(* IEC 61131-3 sources: park-avenue-showroom/park-avenue-showroom/000-main, 28 files *)

(* ---- 000-MAIN.ST ---- *)
VAR_GLOBAL RETAIN
  (*Light groups*)
           (*
           r1_1HallLight01                                  at %R0.0  : bool;
           r2_3LivingroomLight02_07_08                      at %R0.1  : bool; //dimm
           r3_1BalconyLight                                 at %R0.2  : bool;
           r2_2KitchenLight03                               at %R0.3  : bool;
           r2_2KitchenLight04_24                            at %R0.4  : bool;
           r2_1EatingroomLight05_06_23                      at %R0.5  : bool;
           r4_1Bedroom1Light09                              at %R0.6  : bool;
           r5_1Bedroom2Light10_22                           at %R0.7  : bool;
           r5_1Bedroom2Light11                              at %R1.0  : bool;
           r5_1Bedroom2Light12                              at %R1.1  : bool;
           r6_1WardrobeLight13_21                           at %R1.2  : bool;
           r8_1Bathroom2Light14_15_16                       at %R1.3  : bool;
           r7_1Bathroom1Light17_18_19                       at %R1.4  : bool; //dimm
           *)
           supervisorLight_01_08_23_24                      at %R0.0  : bool;
           supervisorLight_02_06_07                         at %R0.1  : bool;
           supervisorLight_balcony                          at %R0.2  : bool;
           supervisorLight_03_04                            at %R0.3  : bool;
           supervisorLight_05                               at %R0.4  : bool;
           supervisorLight_09                               at %R0.5  : bool;
           supervisorLight_10_13_22                         at %R0.6  : bool;
           supervisorLight_11_12_21                         at %R0.7  : bool;
           supervisorLight_14_16                            at %R1.0  : bool;
           supervisorLight_15                               at %R1.1  : bool;
           supervisorLight_17_19                            at %R1.2  : bool;
           supervisorLight_18                               at %R1.3  : bool;

(*Lightgroups mode switches*)
              (*
           r1_1HallLight01_auto                             at %R1.5  : bool;
           r2_3LivingroomLight02_07_08_auto                 at %R1.6  : bool; //dimm
           r2_2KitchenLight03_auto                          at %R1.7  : bool;
           r2_2KitchenLight04_24_auto                       at %R2.0  : bool;
           r2_1EatingroomLight05_06_23_auto                 at %R2.1  : bool;
           r4_1Bedroom1Light09_auto                         at %R2.2  : bool;
           r5_1Bedroom2Light10_auto                         at %R2.3  : bool;
           r5_15Bedroom2Light11_auto                        at %R2.4  : bool;
           r5_15Bedroom2Light12_auto                        at %R2.5  : bool;
           r6_1WardrobeLight13_21_auto                      at %R2.6  : bool;
           r8_1Bathroom2Light14_15_16_auto                  at %R2.7  : bool;
           r7_1Bathroom1Light17_18_19_auto                  at %R3.0  : bool; //dimm
              *)
           supervisorAuto01                                 at %R1.5  : bool; (*Hall*)
           supervisorAuto02                                 at %R1.6  : bool; (*Kitchen*)
           supervisorAuto03                                 at %R1.7  : bool; (*EatingRoom*)
           supervisorAuto04                                 at %R2.0  : bool; (*Bedroom01*)
           supervisorAuto05                                 at %R2.1  : bool; (*Livingroom*)
           supervisorAuto06                                 at %R2.2  : bool; (*Bedroom02*)
           supervisorAuto07                                 at %R2.3  : bool; (*Wardrobe*)
           supervisorAuto08                                 at %R2.4  : bool; (*Bathroom01*)
           supervisorAuto09                                 at %R2.5  : bool; (*Bathroom02*)

(*Blinds Moving Buttons*)
           r2_1EatingroomBlindsUp                           at %R3.1  : bool;
           r2_1EatingroomBlindsDown                         at %R3.2  : bool;
           r2_1EatingroomBlindsStop                         at %R3.3  : bool;
           r4_1Bedroom1BlindsUp                             at %R3.4  : bool;
           r4_1Bedroom1BlindsDown                           at %R3.5  : bool;
           r4_1Bedroom1BlindsStop                           at %R3.6  : bool;
           r5_1Bedroom2BlindsUp                             at %R3.7  : bool;
           r5_1Bedroom2BlindsDown                           at %R4.0  : bool;
           r5_1Bedroom2BlindsStop                           at %R4.1  : bool;

           generalPower                                     at %R4.2  : bool;

(*Floor Heating control*)
           floorHeatingState                                at %R4.3  : bool;

(*Water control*)
           waterState                                       at %R4.4  : bool;
           waterClose                                       at %R4.5  : bool;
           waterOpen                                        at %R4.6  : bool;
           waterAlarmReset                                  at %R4.7  : bool;
           waterAlarm                                       at %R5.0  : bool;

(*Security System*)
           security_arm                                     at %R5.1  : bool;
           security_disarm                                  at %R5.2  : bool;
           security_alarm                                   at %R5.3  : bool;
           security_alarm_reset                             at %R5.4  : bool;
           security_led                                     at %R5.5  : bool;
           security_state                                   at %R5.6  : bool;

(*TV on/off*)
             r2_3_tvOnOff                                   at %R5.7  : bool;
             r2_1_tvOnOff                                   at %R6.0  : bool;

(*Update*)
             updateIridiumProjectFlag                       at %R6.1  : bool;

(*Dimmed groups brightness level*)
           r2_3LivingroomLight02_07_08_level                at %R105  : real;
           r7_1Bathroom1Light17_18_19_level                 at %R109  : real;

(*Blinds position control*)
           r2_1EatingroomBlindsPosition                     at %R113   : real;
           r4_1Bedroom1BlindsPosition                       at %R117   : real;
           r5_1Bedroom2BlindsPosition                       at %R121   : real;

(*Floor Heating control*)
           floorHeatingLevel                                at %R125   : real;

(*AC set temperature*)
           r2_3_GuestRoomACSetTemperature                   at %R129   : real;
           r5_Bedroom2ACSetTemperature                      at %R133   : real;
           r4_Bedroom1ACSetTemperature                      at %R140   : real;
(*AC mode*)
           r2_3_GuestRoomACMode                             at %R137   : usint;
           r5_Bedroom2ACMode                                at %R138   : usint;
           r4_Bedroom1ACMode                                at %R139   : usint;

END_VAR

VAR_GLOBAL CONSTANT
  new : BOOL := false;
  AUTO_MODE_DEFAULT_STATE   : bool := true;
  AUTO_MODE_DEFAULT_TIME    : time := t#150s;
END_VAR

(* ---- fbBlindController.ST ---- *)
FUNCTION_BLOCK fbBlindController
  VAR_INPUT
    timeTo_up_down : time;
    open           : bool r_edge;
    close          : bool r_edge;
    stop           : bool r_edge;
    setPosition    : real;
  END_VAR
  VAR_OUTPUT
    up             : bool;
    down           : bool;
    currentPosition: real:=100;
  END_VAR
  VAR_IN_OUT

  END_VAR
  VAR
    t1             : time;
    timer          : fbTimer;
    direction      : bool;    (*True - UP, False - DOWN*)
    position       : real:=100;
    stopTtigg      : r_trig;
    openTrigg      : r_trig;
    closeTrigg     : r_trig;
  END_VAR
  VAR_TEMP

  END_VAR

  timer();
  if timer.isRun then
    if direction then
      position := position + ((time_to_real(timer.currentTime - t1)/10.)/
                              (time_to_real(timeTo_up_down)/1000.));
    else
      position := position - ((time_to_real(timer.currentTime - t1)/10.)/
                              (time_to_real(timeTo_up_down)/1000.));
    end_if;
    t1 := timer.currentTime;
  else
    t1 := t#0ms;
  end_if;

  currentPosition := position;

  if setPosition>0. then
     if setPosition>currentPosition then
        open:=true;
     end_if;
     if setPosition<currentPosition then
        close:=true;
     end_if;
  end_if;

  if currentPosition <= 0. or currentPosition >= 100. then
     stop:= true;
  end_if;

  if abs(setPosition - currentPosition) <= 0.05 then
     setPosition:=0.;
     stop:= true;
  end_if;

  openTrigg(CLK := open);
  if openTrigg.Q then
    timer(start := true, timeToCount := timeTo_up_down + t#20ms);
    t1 := t#0ms;
    up := true;
    down := false;
    direction := true;
  end_if;

  closeTrigg(CLK := close);
  if closeTrigg.Q then
    timer(start := true, timeToCount := timeTo_up_down + t#20ms);
    t1 := t#0ms;
    up := false;
    down := true;
    direction := false;
  end_if;

  stopTtigg(CLK := stop);
  if stopTtigg.Q then
     up:=false;
     down:=false;
     timer(reset:=true);
     setPosition:=0.;
  end_if;

  timer();
  if timer.isDone then
    timer(reset := true);
    up := false;
    down := false;
  end_if;
END_FUNCTION_BLOCK

(* ---- fbBoolObserver.ST ---- *)
FUNCTION_BLOCK fbBoolObserver
  VAR_INPUT
	  state        : bool;
  END_VAR
  VAR
      prevState : bool;
  END_VAR
  VAR_OUTPUT
      stateChanged : bool;
      rising       : bool;
      falling      : bool;
  END_VAR
  VAR_IN_OUT

  END_VAR
  VAR_TEMP

  END_VAR
      stateChanged := false;
      rising       := false;
      falling      := false;
      if state <> prevState then
         stateChanged := true;
         if state then
            rising := true;
         else
            falling := true;
         end_if;
         prevState := state;
      end_if;
END_FUNCTION_BLOCK

(* ---- fbDataKeeper.st ---- *)
VAR_GLOBAL
    //reader : ReadFromFile; {hidden}
    //writer : WriteToFile;  {hidden}
END_VAR

FUNCTION_BLOCK fbSaveData  {hidden}
  VAR_INPUT
      save     : bool r_edge;
  END_VAR
  VAR_OUTPUT
      idle        : bool := true;
      done        : bool ;
      currentFile : string[20];
  END_VAR
  VAR_IN_OUT
      fullPath    : string[20];
      dataSize    : udint;
      data        : udint;
  END_VAR
  VAR
      lastError: string;
      writer   : WriteToFile;  {hidden}
  END_VAR
  VAR_TEMP
  END_VAR

  done    := false;

  if save then
     idle := false;
     save := false;
  end_if;

  writer( fileName := fullPath,
          srcVar   := data,
          exec     := not idle,
          seek     := 0,
          size     := dataSize);

  if writer.done then
     idle := true;
     done := true;
  end_if;

  if GetLastErr() <> 0 then
     GetLastErrTxt(errCode := GetLastErr(), errMessage := lastError);
  end_if;

  currentFile := fullPath;

END_FUNCTION_BLOCK

FUNCTION_BLOCK fbLoadData  {hidden}
  VAR_INPUT
      load     : bool r_edge;
  END_VAR
  VAR_OUTPUT
      idle        : bool := true;
      done        : bool;
      currentFile : string[20];
  END_VAR
  VAR_IN_OUT
      fullPath    : string[20];
      dataSize : udint;
      data     : udint;
  END_VAR
  VAR
      lastError: string;
      reader   : ReadFromFile; {hidden}
  END_VAR
  VAR_TEMP
  END_VAR

  done    := false;

  if load then
     idle := false;
     load := false;
  end_if;

  reader( fileName := fullPath,
          dstVar   := data,
          exec     := not idle,
          seek     := 0,
          size     := dataSize);

  if reader.done then
     idle := true;
     done := true;
  end_if;

  if GetLastErr() <> 0 then
     GetLastErrTxt(errCode := GetLastErr(), errMessage := lastError);
  end_if;

  currentFile := fullPath;

END_FUNCTION_BLOCK

VAR_GLOBAL RETAIN
    dataSaver  :fbSaveData;    {hidden}
    dataLoader :fbLoadData;    {hidden}
END_VAR

FUNCTION_BLOCK fbDataKeeper
  VAR_INPUT
      path     : string[10];
      fileName : string[10];
      dataSize : udint;
  END_VAR
  VAR_OUTPUT
      load     : bool;
  END_VAR
  VAR_IN_OUT
      data       : udint;
  END_VAR
  VAR
      save     : bool;
      fullPath : string[20];
      init     : bool;
  END_VAR
  VAR_EXTERNAL
      at %s20.3 : bool;
  END_VAR

      fullPath := '/'+ path + '/' +fileName;

      if not init then
         if not FileExists(fileName := fullPath) then
            if not FileExists(fileName := path) then
               DirCreate(dirName := path);
            end_if;
            load := true;
         end_if;
         init := true;
      end_if;

      if not load  then
         if dataLoader.idle then
            dataLoader( load     := true,
                        fullPath := fullPath,
                        dataSize := dataSize,
                        data     := data);
         end_if;
         if dataLoader.done and dataLoader.currentFile = fullPath then
            load := true;
         end_if;
      end_if;

      if %S20.3 and init and load then
         save := true;
      end_if;

      if dataSaver.idle and save  then
         dataSaver( save      := true,
                    fullPath  := fullPath,
                    dataSize  := dataSize,
                    data      := data);
      end_if;
      if dataSaver.done and dataSaver.currentFile = fullPath then
         save     := false;
      end_if;

      dataSaver (data:=data, fullPath := fullPath, dataSize := dataSize);
      dataLoader(data:=data, fullPath := fullPath, dataSize := dataSize);

END_FUNCTION_BLOCK

(* ---- fbFloorHeatingSimple.ST ---- *)
FUNCTION_BLOCK fbFloorHeatingSimple
  VAR_INPUT
       period : time := t#30m;
  END_VAR
  VAR_OUTPUT
      out : bool;
  END_VAR
  VAR_IN_OUT
       state : bool;
       power : real;
  END_VAR
  VAR
       pwmGenerator : PWM;
  END_VAR
  VAR_TEMP
  END_VAR

       pwmGenerator(Enb := true, Per := period, Pls := power, Out =>  out);

       if state then
          out := pwmGenerator.Out;
       else
          out := false;
       end_if;

END_FUNCTION_BLOCK

(* ---- fbGlobalCacheSender.ST ---- *)
TYPE
  irCodesString   :  array[100..150] of string[255];
END_TYPE

FUNCTION_BLOCK fbGlobalCacheSender
  VAR_INPUT
      sendCode : uint;
      channel  : uint;
  END_VAR
  VAR_IN_OUT
      codes   : irCodesString;
  END_VAR
  VAR
      tcpSender : fbSendTo;
      code      : string[255];
      send      : bool;
  END_VAR
      if sendCode <> 0 and (not send) then
         code := codes[sendCode];
         code := code + '$R';
         send           := true;
         sendCode := 0;
      end_if;

      if send then

          tcpSender( chanCode := channel,
                     rq       := not tcpSender.mesSent,
                     lenTx    := len(code),
                     data     := void(code));

          if tcpSender.mesSent then
             send         := false;
          end_if;
      end_if;
END_FUNCTION_BLOCK

(* ---- fbPanel.ST ---- *)
FUNCTION_BLOCK fbPanel
  VAR_INPUT
      button : array[1..6] of fbButtonProcessor;
  END_VAR
  VAR_OUTPUT
      led : array[1..6] of bool;
  END_VAR
  VAR_IN_OUT
  END_VAR
  VAR
  END_VAR
  VAR_TEMP
  END_VAR

    button[1]();
    button[2]();
    button[3]();
    button[4]();
    button[5]();
    button[6]();

END_FUNCTION_BLOCK

(* ---- fbRealObserver.ST ---- *)
FUNCTION_BLOCK fbRealObserver
  VAR_INPUT
	  value        : real;
  END_VAR
  VAR
      prevValue : real;
  END_VAR
  VAR_OUTPUT
      valueChanged : bool;
      rising       : bool;
      falling      : bool;
  END_VAR
      valueChanged := false;
      rising       := false;
      falling      := false;

      if value <> prevValue then
         valueChanged := true;
         if value > prevValue then
            rising := true;
         else
            falling := true;
         end_if;
         prevValue := value;
      end_if;
END_FUNCTION_BLOCK

(* ---- fbSecuritySystem.ST ---- *)
Type
    SecuritySystemState : (init, disarmed, arming, armed, alarming);
    SecurityZoneMode    : (NO,NC);
    SecurityConfig      :
        struct
               exitTime        :time := t#15s;
               enterenceTime   :time := t#15s;
               Z1Mode          :SecurityZoneMode := NC;
               Z2Mode          :SecurityZoneMode := NC;
               Z3Mode          :SecurityZoneMode := NC;
               Z4Mode          :SecurityZoneMode := NC;
               Z5Mode          :SecurityZoneMode := NC;
               KeyBoardEnable  :bool := false;
               KeyBImpulseTime :time := t#1s;
        end_struct;
end_type

FUNCTION_BLOCK fbSecuritySystem
(*
Error codes description:
1 - Can't Armed system because Sabotage alarm is on.
2 - Can't Armed system because one or more zone is broken.
3 - Keypad error.
*)
  VAR_INPUT
    config      :SecurityConfig;
    Z1          :bool; (*Enter/Exit Door.*)
    Z2          :bool; (*Enter/Exit Zone.*)
    Z3          :bool; (*Doors, windows and PIR sensors.*)
    Z4          :bool; (*Other sensors.*)
    Z5          :bool; (*Tamper zone.*)
    keyBoard    :bool; (*relay keypad contact.*)
    arm         :bool r_edge;  (*Security On flag.*)
    disarm      :bool r_edge;  (*Security Off flag.*)
    alarmReset  :bool r_edge;  (*Alarm reset flag.*)
    sabotageReset:bool r_edge; (*Reset sabotege alarm.*)
  END_VAR
  VAR_OUTPUT
    securityState :bool;      (*TRUE when systen armed.*)
    alarm         :bool;      (*Alarm flag.*)
    siren         :bool;      (**)
    ledIndicator  :bool;      (**)
    sabotage      :bool;      (*TRUE when tamper zone was broken until reset by sabotageReset variable.*)
    error         :bool;      (*TRUE when error until next cycle.*)
    errorCode     :usint;     (*Error descrintion code.*)
  END_VAR
  VAR
    state               :SecuritySystemState;
    keyBoardImpulse     :TP;
    keyBoardEvent       :f_trig;
    keyBoardImpulseEnd  :f_trig;
    exitTimer           :ton;
    entranceTimer       :ton;
    ledPulse            :PWM;
    userEnterPassword   :bool;
    armWithoutDelay     :bool;
  END_VAR

//--Zone inverting accordin to their mode (FALSE - normal state)--//
  if config.Z1Mode = NC then
     Z1 := not Z1;
  end_if;

  if config.Z2Mode = NC then
     Z2 := not Z2;
  end_if;

  if config.z3Mode = NC then
     z3 := not z3;
  end_if;

  if config.z4Mode = NC then
     z4 := not z4;
  end_if;

  if config.z5Mode = NC then
     z5 := not z5;
  end_if;

//--General process-//
  if state <> init then
      error := false;

      if config.KeyBoardEnable then
          keyBoardImpulse(IN := not keyBoard, PT := config.KeyBImpulseTime + t#1s);
          keyBoardEvent(CLK := not keyBoard);
          keyBoardImpulseEnd(CLK := keyBoardImpulse.Q);

          userEnterPassword := false;
          userEnterPassword := keyBoardEvent.Q and keyBoardImpulse.Q;

          if keyBoardImpulseEnd.Q and (not keyBoard) then
             error     := true;
             errorCode := 3;
          end_if;
      end_if;

      if Z5 then
         sabotage := true;
      else
         if sabotageReset then
            sabotage := false;
         end_if;
      end_if;
  end_if;

  case state of
    init:
        state := disarmed;

    disarmed:
        if userEnterPassword or arm then
           if (not Z3) and (not Z4) and  (not Z5) and (not sabotage) then
              state := arming;
              if arm then
                 armWithoutDelay := true;
              else
                 armWithoutDelay := false;
              end_if;
           else
              error     := true;
              if sabotage then
                 errorCode := 1;
              else
                 errorCode := 2;
              end_if;
           end_if;
        end_if;
        ledIndicator := false;
        siren        := false;

    arming:
        exitTimer(IN := true, PT := config.exitTime);

        if Z3 or Z4 or Z5 then
           exitTimer(IN := false);
           error     := true;
           if sabotage then
              errorCode := 1;
           else
              errorCode := 2;
           end_if;
           state     := disarmed;
        end_if;

        if exitTimer.Q or armWithoutDelay then
           exitTimer(IN := false);
           if (not Z1) and (not Z2) then
              state := armed;
           else
              error     := true;
              errorCode := 2;
              state     := disarmed;
           end_if;
        end_if;

        ledPulse(Enb := true, Per := t#1s, Pls := 50.0, Out => ledIndicator);

    armed:
        if Z1 then
           entranceTimer.IN := true;
        end_if;

        if (Z2 and not entranceTimer.IN) or Z3 or Z4 or Z5 then
           state := alarming;
        end_if;

        //if (userEnterPassword and entranceTimer.IN) or disarm then
        if userEnterPassword or disarm then
           state := disarmed;
           entranceTimer(IN := false);
        end_if;

        entranceTimer(PT := config.enterenceTime);
        if entranceTimer.Q then
           entranceTimer(IN := false);
           state := alarming;
        end_if;

        if entranceTimer.IN then
           ledPulse(Enb := true, Per := t#1s, Pls := 50.0, Out => ledIndicator);
        else
           ledIndicator := true;
        end_if;
        siren := false;

    alarming:
        siren := true;
        ledPulse(Enb := true, Per := t#2s, Pls := 75.0, Out => ledIndicator);
        if alarmReset then
           state := armed;
        end_if;

        if userEnterPassword or disarm then
           state := disarmed;
           entranceTimer(IN := false);
        end_if;

  end_case;

  if state <> init then
       if state = alarming then
         alarm := true;
      else
         alarm := false;
      end_if;

      if state = armed then
         securityState := true;
      end_if;

      if state = disarmed then
         securityState := false;
      end_if;
  end_if;

END_FUNCTION_BLOCK

(* ---- fbTimer.ST ---- *)
FUNCTION_BLOCK fbTimer
  VAR_INPUT
      start      : bool r_edge;
      reset      : bool r_edge;
      timeToCount: time;
  END_VAR
  VAR_OUTPUT
      isRun : bool;
      isDone: bool;
      currentTime : time;
  END_VAR
  VAR_IN_OUT
  END_VAR
  VAR
      timer: TON;
  END_VAR
  VAR_TEMP
  END_VAR

         if start and not isRun then
            timer.IN := true;
            start    := false;
            isRun    := true;
            isDone   := false;
            timer.PT := timeToCount;
         end_if;

         if start and isRun then
            timer(IN :=false);
            timer(IN :=true);
         end_if;

         if isRun then
            timer();
            if timer.ET>=timer.PT then
               isDone:=true;
               isRun :=false;
               timer.IN:=false;
               timer();
            end_if;
         end_if;

         if reset then
            timer.IN:=false;
            isDone:=false;
            isRun:=false;
            timer();
         end_if;

         timer();
         currentTime:=timer.ET;
END_FUNCTION_BLOCK

(* ---- prgNotifications.ST ---- *)
FUNCTION_BLOCK fbBoolObserver
  VAR_INPUT
      in : bool;
  END_VAR
  VAR
      prevState : bool;
  END_VAR
  VAR_OUTPUT
      stateChanged : bool;
      state        : bool;
      rising       : bool;
      falling      : bool;
  END_VAR
      stateChanged := false;
      rising       := false;
      falling      := false;
      state        := in;
      if state <> prevState then
         stateChanged := true;
         if state then
            rising := true;
         else
            falling := true;
         end_if;
         prevState := state;
      end_if;
END_FUNCTION_BLOCK

FUNCTION_BLOCK fbRealObserver
  VAR_INPUT
      in : ptr_to real;
  END_VAR
  VAR
      prevValue : real;
  END_VAR
  VAR_OUTPUT
      valueChanged : bool;
      value        : real;
      rising       : bool;
      falling      : bool;
  END_VAR
      valueChanged := false;
      rising       := false;
      falling      := false;
      value        := in^;

      if value <> prevValue then
         valueChanged := true;
         if value > prevValue then
            rising := true;
         else
            falling := true;
         end_if;
         prevValue := value;
      end_if;
END_FUNCTION_BLOCK

(* ---- RalayAndDimmer.ST ---- *)
type
    motionSensorMode: (null, NO, NC);
    doorSensorMode:   (null, NO, NC);
    motionSensor:
        struct
            state:bool;
            mode :motionSensorMode;
        end_struct;
    doorSensor:
        struct
            state:bool;
            mode :doorSensorMode;
        end_struct;
end_type

FUNCTION_BLOCK fbAutoRelay
  VAR_IN_OUT
           //trigButton      : bool ;                  (**)
           //autoMode        : bool :=true;
  END_VAR
  VAR_INPUT
           Sensor_Door      : doorSensor;   (**)
           Sensor_Motion    : motionSensor; (**)

           autoMode      : bool ;                    (**)
           nightMode     : bool ;                    (**)

           forgetMode    : bool :=false;             (**)

           anyLightOn             : bool ;           (**)
           anyLightChanged        : bool ;           (**)

           timeAfterDoorOpenClose : time :=t#1m;     (**)
           timeAfterMotionDetect  : time :=t#10m;     (**)
           timeAfterLastAction    : time :=t#1m;     (**)
           setState               : bool ;           (**)
  END_VAR
  VAR_OUTPUT
           personLeft   : bool ;                     (**)
           forget       : bool ;                     (**)
           stateChanged : bool ;                     (**)
           state        : bool ;                     (**)
  END_VAR
  VAR
           timerAfterDoorOpened     : fbTimer;
           timerAfterDoorClosed     : fbTimer;
           timerAfterMotionDetected : fbTimer;
           timerAfterLastAction     : fbTimer;

           doorSensRise        : r_trig;
           doorSensFall        : f_trig;
           doorClosed          : bool;
           doorOpened          : bool;
           motionSensRise      : r_trig;
           motionSensFall      : f_trig;
           motionDetected      : bool;
           motionEnd           : bool;
           nightModeOff        : f_trig;
  END_VAR

        (*Refresh outputs.*)
        stateChanged:=false;
        personLeft  :=false;
        forget      :=false;

        nightModeOff(CLK := nightMode);
        if nightModeOff.Q then
           timerAfterDoorOpened    (reset := true);
           timerAfterDoorClosed    (reset := true);
           timerAfterMotionDetected(reset := true);
           if autoMode then
              setState:=false; end_if;
        end_if;

        (*Auto*)
        if autoMode and nightMode then
           (*Process move sensor.*)
           motionSensRise(CLK := Sensor_Motion.state);
           motionSensFall(CLK := Sensor_Motion.state);
           case Sensor_Motion.mode of
                NO:
                   motionDetected := motionSensRise.Q;
                   motionEnd      := motionSensFall.Q;
                NC:
                   motionDetected := motionSensFall.Q;
                   motionEnd      := motionSensRise.Q;
           end_case;
           (*Process door sensor.*)
           case Sensor_Door.mode of
                NO:
                   doorSensRise(CLK := Sensor_Door.state, Q => doorOpened);
                   doorSensFall(CLK := Sensor_Door.state, Q => doorClosed);
                NC:
                   doorSensRise(CLK := Sensor_Door.state, Q => doorClosed);
                   doorSensFall(CLK := Sensor_Door.state, Q => doorOpened);
           end_case;
           (*Timers process.*)
           timerAfterDoorOpened     (timeToCount :=timeAfterDoorOpenClose);
           timerAfterDoorClosed     (timeToCount :=timeAfterDoorOpenClose);
           timerAfterMotionDetected (timeToCount :=timeAfterMotionDetect);
           (*Door opened/closed logic.*)
           (*Door opened.*)
           if doorOpened and not anyLightOn then
              setState:=true;
              timerAfterDoorOpened( start := true);
           end_if;
           timerAfterDoorOpened();
           if timerAfterDoorOpened.isDone then
              setState :=false;
              timerAfterDoorOpened(reset := true);
           end_if;
           (*Door closed.*)
           if doorClosed then
              timerAfterDoorClosed( start := true);
           end_if;
           if timerAfterDoorClosed.isDone then
              setState  :=false;
              personLeft:=true;
              timerAfterDoorClosed(reset := true);
           end_if;
           (*Motion detecion logic.*)
           (*Motion detected.*)
           if motionDetected then
              if not anyLightOn then
                 setState := true;
//                 timerAfterMotionDetected(start := true);
              end_if;
              timerAfterDoorOpened    (reset := true);
              timerAfterDoorClosed    (reset := true);
           end_if;
           (*Motion end.*)
           if motionEnd then
              timerAfterMotionDetected(start := true);
           end_if;
           if timerAfterMotionDetected.isDone then
              setState:=false;
              timerAfterMotionDetected(reset := true);
           end_if;
        end_if;

        (*Forget mode.*)
        if forgetMode then
           timerAfterLastAction(timeToCount := timeAfterLastAction);
           if motionDetected then
              timerAfterLastAction(start := true);
           end_if;
           if timerAfterLastAction.isDone then
              timerAfterLastAction(reset:=true);
              forget:=true;
           end_if;
           if anyLightChanged then
              timerAfterLastAction(reset:=true);
              timerAfterLastAction(start:=true);
           end_if;;
        end_if;

        (*Set state.*)
        if setState<>state then
           stateChanged:= true;
           state       := setState;
        end_if;
END_FUNCTION_BLOCK

FUNCTION_BLOCK fbManualRelay
  VAR_IN_OUT
           trigButton          : bool ; (*Button for trigger control.*)
  END_VAR
  VAR_INPUT
           setState            : bool ; (*Turn on/off channel.*)
  END_VAR
  VAR
           trigButtonOff   : f_trig;
           trigButtonOn    : r_trig;
  END_VAR
  VAR_OUTPUT
           stateChanged : bool  ;           (*State changed flag.    *)
           state        : bool ;            (*Current state of relay.*)
  END_VAR
        (*Refresh outputs.*)
        stateChanged:=false;

        trigButtonOn (CLK := trigButton);
        trigButtonOff(CLK := trigButton);

        if trigButtonOn.Q  then
           setState:=true;
        end_if;

        if trigButtonOff.Q then
           setState:=false;
        end_if;

        if setState<>state then
           stateChanged := true;
           state        := setState;
           trigButton   := state;
        end_if;

END_FUNCTION_BLOCK

function_block fbButtonProcessor
    var_input
        btn          :  bool; (*Pointer to Button*)
        longPressTime: time := t#1000ms;       (*Long press time detect.*)
    end_var
    var_in_out
    end_var
    var_output
        longPress  :bool;                     (*Long press flag.*)
        shortPress :bool;                     (*Short press flag.*)
        btnPressed :bool;                     (*Event flag on button pressed.*)
        btnReleased:bool;                     (*Event flag on button released.*)
        btnState   :bool;                     (*Button state.*)
        longPressAndHold:bool;                (*Long press and hold flag.*)
    end_var
    var
        btnPrevState  :bool;
        timer         :fbTimer;
    end_var
    var
    end_var
        (*Refresh outputs.*)
        longPress  :=false;
        shortPress :=false;
        btnPressed :=false;
        btnReleased:=false;
        btnState   :=btn;
        (*Button event detection.*)
        timer(timeToCount := longPressTime);
        if btn <> btnPrevState then
           (*Button status changed.*)
           btnPrevState := btn;
           if btn then
              (*Button pressed.*)
              btnPressed:=true;
              if not timer.isRun then
                 timer.start:=true;
                 timer();
              end_if;
           else
              (*Button Released.*)
              btnReleased:=true;
              if timer.isRun then
                 timer.reset := true;
                 timer();
                 shortPress:=true;
              end_if;
           end_if;
        end_if;
        if timer.isDone then
           (*Time out.*)
           timer.reset := true;
           timer();
           longPress:=true;
        end_if;

        if longPress then
           longPressAndHold:=true;
        end_if;

        if btnReleased then
           longPressAndHold := false;
        end_if;

end_function_block

function_block fbManualDimm
    var_input
        btn      : bool;                       (*Pointer to button processor.*)
        minValue : real:=20.0;                 (*Minimum value of channel.*)
        maxValue : real:=100.0;                (*Maximum value of channel.*)
        dimmSpeed: real:=25.0;                 (*Up/Down dimming speed, %/sec.*)
        setValue : real;                       (**)
        setState : bool;                       (*Turn on/off channel like relay. Set to levels like short press.*)
    end_var
    var_in_out
        slider    :real;                       (*Slider in % in range from minValue to maxValue.*)
        trigButton:bool;                       (*Button for trigger contol.*)
    end_var
    var_output                                 (*Current value of channel.*)
        value       :real;
        valueChanged:bool;
        state       :bool;
        stateChanged:bool;
    end_var
    var
        direction :real:=1.0;
        userValue :real;
        dimming   :bool;
        timer     :TON;
        cycleTime :time;
        prevTime  :time;
        step      :real;
        init      :bool;
        prevValue :real;
        prevSetValue:real;
        prevSlider:real;
        buttonProcessor : fbButtonProcessor;
    end_var
    var_temp

    end_var
        (*Init block.*)
        if not init then
           init:=true;
           userValue:=maxValue;
        end_if;

        buttonProcessor(btn := btn);

        (*Calc 1% in current range.*)
        if minValue<20. then
           minValue:=20.; end_if;
        step:=((maxValue-minValue)/100.);

        (*Reset outputs.*)
        valueChanged:=false;
        stateChanged:=false;

        (*Set value by setValue variable.*)
        if setValue<>prevSetValue then
           if setValue=0.0 then
              value:=0.0;
           elsif setValue=1.0 then
              value := minValue;
           else
              value := minValue + (step*setValue);
           end_if;
        end_if;

        (*Set value by slider.*)
        if slider<>prevSlider then
           if slider=0.0 then
              value:=0.0;
           elsif slider=1.0 then
              value := minValue;
           else
              value := minValue + (step*slider);
           end_if;
        end_if;

        (*On/Off channel.*)
        (*On/Off by impulse button.*)
        if buttonProcessor.shortPress then
           if value >= minValue then
              userValue := value;
              value  := 0.0;
           else
              value := userValue;
           end_if;
        end_if;
        (*On/Off by setState variable.*)
        if setState<>state then
           if setState then
              value:=userValue;
           else
              value:=0.0;
           end_if;
        end_if;
        (*On/Off by triggButton variable.*)
        if trigButton <> state then
           if trigButton then
              value:=userValue;
           else
               value:=0.0;
           end_if;
        end_if;

        (*Dimming.*)
        timer(IN := buttonProcessor.longPressAndHold , PT := t#100s);
        cycleTime:=SUB_TIME(IN1 := timer.ET, IN2 := prevTime);
        prevTime:=timer.ET;

        if buttonProcessor.longPressAndHold then
           dimming:=true;
           value:=value + (direction * (step * dimmSpeed * (TIME_TO_REAL(cycleTime)/1000.)));
           if value > maxValue then
              value := maxValue; end_if;
           if value < minValue then
              value := minValue; end_if;
        end_if;

        (*End_dimming.*)
        if dimming and buttonProcessor.btnReleased then
           dimming   := false;
           direction := direction*(-1.0);
           userValue := value;
        end_if;

         (*Update slider and local variables.*)
         if value=0.0 then
            slider:=0.0;
         elsif value=minValue then
            slider:=1.0;
         else
            slider:=((value-minValue)/step);
            if slider>100. then
               slider:=100.; end_if;
         end_if;
         prevSlider  :=slider;
         setValue    :=slider;
         prevSetValue:=slider;
         trigButton  := REAL_TO_BOOL(value);
         setState    := trigButton;

         (*Update outputs.*)
         if state <> REAL_TO_BOOL(value) then
            stateChanged:=true;
            state := REAL_TO_BOOL(value);
         end_if;
         if value <> prevValue then
            prevValue    :=value;
            valueChanged :=true;
         end_if;
end_function_block

(* ---- WaterLeakegeControl.ST ---- *)
TYPE
  WaterSensorModeType : (NO, NC); (*NO: Alarm when input is TRUE. NC: alarm when input is FALSE.*)
  WaterValveModeType  : (NO, NC); (*NO: Valve is open when output = FALSE; NC: Valve is open when output = TRUE *)
  WaterLeakegeControlConfig:
    STRUCT
      sensorMode                : WaterSensorModeType := NO;
      valveMode                 : WaterValveModeType  := NO;
      timeTreshold              : time           := t#5s;
      waterOnSendorsTimeoutTime : time           := t#10m;
    END_STRUCT;
END_TYPE

FUNCTION_BLOCK fbWaterLeakegeControl
  VAR_INPUT
  //--Inputs--//
      sensor     : bool ;                     (*Water Leakege Sensor.*)
  //--Commands--//
      openWater  : bool r_edge;               (*Flag to open water if it possible.*)
      closeWater : bool r_edge;               (*Flag to close water.*)
      alarmReset : bool r_edge;               (*Flag to reset alarm.*)
  //--Configuration variables--//
      config     : WaterLeakegeControlConfig; (*Zone configuration.*)
      autoControl: bool := true;
  END_VAR
  VAR_OUTPUT
      valve      : bool;                      (*Valve.*)
      alarm      : bool;                      (*True when water was closed by sensor until not reset.*)
  END_VAR
  VAR_IN_OUT
      waterState : bool                       (*TRUE = Water is open.*);
  END_VAR
  VAR
      waterOnSensor         : bool;
      timeTreshold          : ton;
      waterOnSendorsTimeout : tp;
      timeOut               : f_trig;
  END_VAR

  case config.sensorMode of
       NO: waterOnSensor := sensor;
       NC: waterOnSensor := not sensor;
  end_case;

  if openWater then
     waterState := true;
  end_if;

  if closeWater then
     waterState := false;
  end_if;

  if alarmReset then
     alarm := false;
     waterOnSendorsTimeout(IN := false); // timer call to reset
     waterOnSendorsTimeout.IN := true;
  end_if;

  timeTreshold(IN := waterOnSensor, PT := config.timeTreshold);
  waterOnSendorsTimeout(PT := config.waterOnSendorsTimeoutTime);
  timeOut(CLK := waterOnSendorsTimeout.Q);

  if timeTreshold.Q or (timeOut.Q and waterOnSensor) then
     alarm := true;
  end_if;

  if alarm and autoControl then
     waterState := false;
  end_if;

  if waterState and alarm then
     waterState := false;
  end_if;

  case config.valveMode of
       NO: valve := not waterState;
       NC: valve := waterState;
  end_case;

END_FUNCTION_BLOCK

(* ---- prgBalconyLight.ST ---- *)
PROGRAM prgBalconyLight
  VAR_INPUT
  END_VAR
  VAR_OUTPUT
  END_VAR
  VAR
      Lamp1     : fbManualRelay;

      button    : fbButtonProcessor;

      init      : bool;
  END_VAR
  VAR_TEMP
  END_VAR

  if not init then
     init := true;
  end_if;

  button(btn :=button_04_1);

  if button.shortPress then
     Lamp1.setState:= not Lamp1.state;
  end_if;

  lamp1(
        trigButton := supervisorLight_balcony,
        state      => light_balcony
        );

  if generalPowerObserver.falling then
     Lamp1.setState := false;
  end_if;

END_PROGRAM

(* ---- prgBathroom1Light.ST ---- *)
PROGRAM prgBathroom1Light
  VAR_INPUT
  END_VAR
  VAR_OUTPUT
  END_VAR
  VAR

      Lamp1,
      Lamp2     : fbManualRelay;

      Auto8      : fbAutoRelay;

      button1,
      button2   : fbButtonProcessor;

      init      : bool;

  END_VAR
  VAR_TEMP
  END_VAR

  if not init then
     supervisorAuto08                 := AUTO_MODE_DEFAULT_STATE;
     Auto8.timeAfterMotionDetect       := AUTO_MODE_DEFAULT_TIME;
     Auto8.Sensor_Motion.mode          := NC;
     Auto8.nightMode                   := true;

     init := true;
 end_if;

 (*Lamp1*)
  button1(btn := button_15_1_16_1);

  if button1.shortPress then
     Lamp1.setState := not Lamp1.state;
  end_if;

  Lamp1(trigButton := supervisorLight_17_19);

  light_17_19_level := BOOL_TO_REAL(Lamp1.state) * 100.;

  Auto8(Sensor_Motion.state   := msensor08,
        autoMode              := supervisorAuto08);

  if Auto8.stateChanged then
     Lamp1.setState := Auto8.state;
  end_if;

  (*Lamp2*)
  button2(btn := button_15_2_16_2);

  if button2.shortPress then
     Lamp2.setState := not Lamp2.state;
  end_if;

  Lamp2(trigButton := supervisorLight_18);

  light_18_mirror := Lamp2.state;

  if generalPowerObserver.falling then
     Lamp1.setState := false;
     Lamp2.setState := false;
  end_if;

END_PROGRAM

(* ---- prgBathroom2Light.ST ---- *)
PROGRAM prgBathroom2Light
 VAR_INPUT
  END_VAR
  VAR_OUTPUT
  END_VAR
  VAR
      Lamp1,
      Lamp2     : fbManualRelay;

      Auto9     : fbAutoRelay;

      button1,
      button2   : fbButtonProcessor;

      init      : bool;

      //kostyl    :R_TRIG;

  END_VAR
  VAR_TEMP
  END_VAR

  if not init then
     supervisorAuto09                  := AUTO_MODE_DEFAULT_STATE;
     Auto9.timeAfterMotionDetect       := AUTO_MODE_DEFAULT_TIME;
     Auto9.Sensor_Motion.mode          := NC;
     Auto9.nightMode                   := true;

     init := true;
 end_if;

 (*Lamp1*)
  button1(btn := button_20_1_21_1);

  if button1.shortPress then
     Lamp1.setState := not Lamp1.state;
  end_if;

  //эта штука появилась тут из-за того, что нужно было
  //добавить в сценарий "пришел домой" включение света в СУ2
  //а Юрко не нашел кода, который этот сценарий реализует
  //kostyl(CLK := generalPower);
  if generalPowerObserver.rising Then
     supervisorLight_14_16 := true;
  End_if;

  Lamp1(trigButton := supervisorLight_14_16);

  light_14_16 := Lamp1.state;

  Auto9(Sensor_Motion.state   := msensor09,
        autoMode              := supervisorAuto09);

  if Auto9.stateChanged then
     Lamp1.setState := Auto9.state;
  end_if;

  (*Lamp2*)
  button2(btn := button_20_2_22_1);

  if button2.shortPress then
     Lamp2.setState := not Lamp2.state;
  end_if;

  Lamp2(trigButton := supervisorLight_15);

  light_15 := Lamp2.state;

  if generalPowerObserver.falling then
     Lamp1.setState := false;
     Lamp2.setState := false;
  end_if;

END_PROGRAM

(* ---- prgBedroom1Light.ST ---- *)
PROGRAM prgBedroom1Light
  VAR_INPUT
  END_VAR
  VAR_OUTPUT
  END_VAR
  VAR
      Lamp1     : fbManualRelay;

      Auto4      : fbAutoRelay;

      button    : fbButtonProcessor;

      init      : bool;
  END_VAR
  VAR_TEMP
  END_VAR

  if not init then

     supervisorAuto04                := AUTO_MODE_DEFAULT_STATE;
     Auto4.timeAfterMotionDetect     := AUTO_MODE_DEFAULT_TIME;
     Auto4.Sensor_Motion.mode        := NC;
     Auto4.nightMode                 := true;

     init                           := true;
  end_if;

  button(btn:= button_07_1_08_1);

  if button.shortPress then
     lamp1.setState := not lamp1.state;
  end_if;

  lamp1( trigButton := supervisorLight_09,
         state      =>  light_09
         );

  Auto4(Sensor_Motion.state   := msensor04,
        autoMode              := supervisorAuto04);

  if Auto4.stateChanged then
     Lamp1.setState := Auto4.state;
  end_if;

  if generalPowerObserver.falling then
     Lamp1.setState := false;
  end_if;

END_PROGRAM

(* ---- prgBedroom2Light.ST ---- *)
PROGRAM prgBedroom2Light
  VAR_INPUT
  END_VAR
  VAR_OUTPUT
  END_VAR
  VAR
      Lamp1     : fbManualRelay;
      Lamp2     : fbManualRelay;

      button1   :fbButtonProcessor;
      button2   :fbButtonProcessor;

      Auto6,
      Auto7      : fbAutoRelay;

      init      : bool;
  END_VAR
  VAR_TEMP
  END_VAR

  if not init then
     supervisorAuto06               := AUTO_MODE_DEFAULT_STATE;
     supervisorAuto07               := AUTO_MODE_DEFAULT_STATE;
     Auto6.timeAfterMotionDetect    := AUTO_MODE_DEFAULT_TIME;
     Auto7.timeAfterMotionDetect    := AUTO_MODE_DEFAULT_TIME;
     Auto6.Sensor_Motion.mode       := NC;
     Auto7.Sensor_Motion.mode       := NC;
     Auto6.nightMode                := true;
     Auto7.nightMode                := true;

     init := true;
  end_if;

  (*Lamp1*)
  button1(btn := button_09_1_10_2_17_1);

  if button1.shortPress then
     Lamp1.setState := not Lamp1.state;
  end_if;

  Lamp1(trigButton := supervisorLight_10_13_22);

  light_10_13_22 := Lamp1.state;

  Auto6(Sensor_Motion.state   := msensor06,
        autoMode              := supervisorAuto06);

  if Auto6.stateChanged then
     Lamp1.setState := Auto6.state;
  end_if;

(*Lamp2*)
  button2(btn := button_09_2_09_3_11_1_12_1_13_1_14_1_17_2);

  if button1.shortPress then
     Lamp2.setState := not Lamp2.state;
  end_if;

  Lamp2(trigButton := supervisorLight_11_12_21);

  light_11_12_21 := Lamp2.state;

  Auto7(Sensor_Motion.state   := msensor07,
        autoMode              := supervisorAuto07);

  if Auto7.stateChanged then
     Lamp2.setState := Auto7.state;
  end_if;

  if generalPowerObserver.falling then
     Lamp1.setState := false;
     Lamp2.setState := false;
  end_if;

END_PROGRAM

(* ---- prgEatingroomLight.ST ---- *)
PROGRAM prgEatingroomLight
  VAR_INPUT
  END_VAR
  VAR_OUTPUT
  END_VAR
  VAR

      Lamp1               : fbManualRelay;

      Auto3               : fbAutoRelay;

      buttonUp,
      buttonDown
      (*button*)          : fbButtonProcessor;

      blind               : fbBlindController;

      initTimer           : ton;
      init                : bool;

  END_VAR
  VAR_TEMP
  END_VAR

  if not init then

     supervisorAuto03                        := AUTO_MODE_DEFAULT_STATE;
     Auto3.timeAfterMotionDetect             := AUTO_MODE_DEFAULT_TIME;
     Auto3.Sensor_Motion.mode                := NC;
     Auto3.nightMode                         := true;

     blind.timeTo_up_down                   := t#38000ms;

     //MODULE4_OUT.DO3                        := true; //Типа чтобы штора после старта была открыта
     initTimer( IN := true,
                PT := blind.timeTo_up_down);
     if initTimer.Q then
        init := true;
     end_if;
  else

      blind( //up            => MODULE4_OUT.DO3,
             //down          => MODULE4_OUT.DO4,

             position      := r2_1EatingroomBlindsPosition,

             open          := r2_1EatingroomBlindsUp OR buttonUp.shortPress,
             close         := r2_1EatingroomBlindsDown OR buttonDown.shortPress,
             stop          := r2_1EatingroomBlindsStop);

      r2_1EatingroomBlindsUp    := false;
      r2_1EatingroomBlindsDown  := false;
      r2_1EatingroomBlindsStop  := false;
  end_if;

  (*Lamp1*)
  if panel.button[3].shortPress then
     Lamp1.setState := not Lamp1.state;
  end_if;

  lamp1( trigButton := supervisorLight_05,
         state      => light_05
         );

  panel.led[3]:= Lamp1.state;

  Auto3(Sensor_Motion.state   := msensor03,
        autoMode              := supervisorAuto03);

  if Auto3.stateChanged then
     Lamp1.setState := Auto3.state;
  end_if;

  if generalPowerObserver.falling then
     Lamp1.setState := false;
  end_if;

END_PROGRAM

(* ---- prgFloorHeating.ST ---- *)
PROGRAM prgFloorHeating
  VAR_INPUT
  END_VAR
  VAR_OUTPUT
  END_VAR
  VAR

      termostat : fbFloorHeatingSimple;

  END_VAR
  VAR_TEMP
  END_VAR

      termostat( period := T#30m,
                 state  := floorHeatingState,
                 power  := floorHeatingLevel,
                 //out    =>
                 );

END_PROGRAM

(* ---- prgHallLight.ST ---- *)
PROGRAM prgHallLight
  VAR_INPUT
  END_VAR
  VAR_OUTPUT
  END_VAR
  VAR
      Lamp1     : fbManualRelay;

      Auto1     : fbAutoRelay;

      button    : fbButtonProcessor;

      init      : bool;
  END_VAR
  VAR_TEMP
  END_VAR

  if not init then

     supervisorAuto01               := AUTO_MODE_DEFAULT_STATE;
     Auto1.timeAfterMotionDetect    := AUTO_MODE_DEFAULT_TIME;
     Auto1.Sensor_Motion.mode       := NC;
     Auto1.nightMode                := true;

     init := true;
  end_if;

  if panel.button[1].shortPress then
     Lamp1.setState := not Lamp1.state;
  end_if;

  lamp1( trigButton := supervisorLight_01_08_23_24,
         state      => light_01_08_23_24
         );

  panel.led[1]:= Lamp1.state;

  Auto1( Sensor_Motion.state   := msensor01,
        autoMode              := supervisorAuto01
        );

  if Auto1.stateChanged then
     Lamp1.setState := Auto1.state;
  end_if;

  if generalPowerObserver.falling then
     Lamp1.setState := false;
  end_if;

END_PROGRAM

(* ---- prgKitchenLight.ST ---- *)
PROGRAM prgKitchenLight
   VAR_INPUT
  END_VAR
  VAR_OUTPUT
  END_VAR
  VAR
      Lamp1     : fbManualRelay;

      Auto2     : fbAutoRelay;

      init      : bool;
  END_VAR
  VAR_TEMP
  END_VAR

  if not init then
     supervisorAuto02               := AUTO_MODE_DEFAULT_STATE;
     Auto2.timeAfterMotionDetect    := AUTO_MODE_DEFAULT_TIME;
     Auto2.Sensor_Motion.mode       := NC;
     Auto2.nightMode                := true;
     init := true;
  end_if;

  if panel.button[2].shortPress then
     Lamp1.setState := not Lamp1.state;
  end_if;

  lamp1( trigButton := supervisorLight_03_04,
         state      => light_03_04
         );

  panel.led[2]:= Lamp1.state;

  Auto2( Sensor_Motion.state   := msensor02,
        autoMode               := supervisorAuto02
        );

  if Auto2.stateChanged then
     Lamp1.setState := Auto2.state;
  end_if;

  if generalPowerObserver.falling then
     Lamp1.setState := false;
  end_if;

END_PROGRAM

(* ---- prgLivingroomLight.ST ---- *)
PROGRAM prgLivingroomLight
  VAR_INPUT
  END_VAR
  VAR_OUTPUT
  END_VAR
  VAR
      Lamp1     : fbManualRelay;
      Auto5     : fbAutoRelay;

      init      : bool;
  END_VAR
  VAR_TEMP
  END_VAR

  if not init then

     supervisorAuto05                   := AUTO_MODE_DEFAULT_STATE;
     Auto5.timeAfterMotionDetect        := AUTO_MODE_DEFAULT_TIME;
     Auto5.Sensor_Motion.mode           := NC;
     Auto5.nightMode                    := true;

     init := true;
 end_if;

  if panel.button[4].shortPress then
     Lamp1.setState := not Lamp1.state;
  end_if;

  Lamp1(trigButton :=supervisorLight_02_06_07,
                   state => light_02_06_07);

  panel.led[4]:= Lamp1.state;

  Auto5(Sensor_Motion.state   := msensor05,
        autoMode              := supervisorAuto05);

  if Auto5.stateChanged then
     lamp1.setState := Auto5.state;
  end_if;

  if generalPowerObserver.falling then
     Lamp1.setState := false;
  end_if;

END_PROGRAM

(* ---- prgLivingRoomMedia.ST ---- *)
VAR_GLOBAL CONSTANT
  TV_ON       : uint := 100;
  TV_OFF      : uint := 101;
  PLAYER_ON   : uint := 102;
  PLAYER_OFF  : uint := 103;
  RECEIVER_ON : uint := 104;
  RECEIVER_OFF: uint := 105;
END_VAR

PROGRAM prgLivingRoomMedia
  VAR_INPUT
  END_VAR
  VAR_OUTPUT
  END_VAR
  VAR
      //generalPowerObserber     : fbBoolObserver;
      clock                 : fbTick;
      allOnState  : usint;
      allOffState : usint;
      init : bool;
  END_VAR
  VAR_TEMP
  END_VAR

  if not init then

    globalCacheCodes[TV_ON]        := 'sendir,1:1,1,36000,1,1,32,32,64,31,32,32,32,32,32,32,32,32,32,63,32,32,32,32,32,32,32,32,32,32,32,3600';
    globalCacheCodes[TV_OFF]       := 'sendir,1:1,1,36000,1,1,32,32,64,31,32,32,32,32,32,32,32,32,32,63,32,32,32,32,32,32,64,63,32,3600';
    globalCacheCodes[PLAYER_ON]    := 'sendir,1:1,1,38000,1,1,341,169,21,21,21,21,21,63,21,63,21,63,21,63,21,63,21,21,21,63,21,63,21,21,21,21,21,21,21,21,21,21,21,63,21,21,21,63,21,63,21,21,21,63,21,63,21,63,21,63,21,63,21,21,21,21,21,63,21,21,21,21,21,21,21,21,21,1515,341,85,21,3800';
    globalCacheCodes[PLAYER_OFF]   := 'sendir,1:1,1,38000,1,1,341,169,21,21,21,21,21,63,21,63,21,63,21,63,21,63,21,21,21,63,21,63,21,21,21,21,21,21,21,21,21,21,21,63,21,63,21,63,21,63,21,21,21,63,21,63,21,63,21,63,21,21,21,21,21,21,21,63,21,21,21,21,21,21,21,21,21,1515,341,85,21,3800';
    globalCacheCodes[RECEIVER_ON]  := 'sendir,1:2,1,38000,1,1,341,169,21,20,21,20,21,20,21,20,21,20,21,20,21,20,21,63,21,20,21,20,21,20,21,20,21,63,21,63,21,63,21,20,21,20,21,20,21,20,21,20,21,63,21,20,21,63,21,63,21,63,21,63,21,63,21,63,21,20,21,63,21,20,21,20,21,1513,341,84,21,3800';
    globalCacheCodes[RECEIVER_OFF] := 'sendir,1:2,1,38000,1,1,341,169,21,20,21,20,21,20,21,20,21,20,21,20,21,20,21,63,21,20,21,20,21,20,21,20,21,63,21,63,21,63,21,20,21,63,21,63,21,63,21,63,21,63,21,20,21,20,21,63,21,20,21,20,21,20,21,20,21,20,21,63,21,63,21,20,21,1517,341,85,21,3800';

  end_if;

  //generalPowerObserber(state := generalPower);

  if panel.button[5].shortPress then
     allOnState := 1;
  end_if;

  if panel.button[6].shortPress  or generalPowerObserver.falling then
     allOffState := 1;
  end_if;

  clock(IN := true, PT := T#1000ms);

  if clock.Q then
      case allOnState of
          1:  allOnState := 2; //blank call
          2:
              globalCache.sendCode := TV_ON;
              allOnState := 3;
          3:
              globalCache.sendCode := PLAYER_ON;
              allOnState := 4;
          4:
              globalCache.sendCode := RECEIVER_ON;
              allOnState := 0;
      end_case;

      case allOffState of
          1:  allOffState := 2;
          2:
              globalCache.sendCode := TV_OFF;
              allOffState := 3;
          3:
              globalCache.sendCode := PLAYER_OFF;
              allOffState := 4;
          4:
              globalCache.sendCode := RECEIVER_OFF;
              allOffState := 0;
      end_case;
  end_if;

END_PROGRAM

(* ---- prgMain.ST ---- *)
VAR_GLOBAL
    globalCache : fbGlobalCacheSender;
    globalCacheCodes : irCodesString;
    generalPowerObserver : fbBoolObserver;
    panel : fbPanel;
END_VAR

PROGRAM prgMain
  VAR_INPUT
  END_VAR
  VAR_OUTPUT
  END_VAR
  VAR
         init       : bool;

         generalPowerButton   : fbButtonProcessor;

  END_VAR
  VAR_TEMP
  END_VAR

   if not init then
         generalPower      := true;
         electricitySwitch := true;

         generalPowerButton.longPressTime := T#2s;

         r2_3_GuestRoomACSetTemperature := 23.0;
         r5_Bedroom2ACSetTemperature := 20.0;
         r4_Bedroom1ACSetTemperature := 20.0;

         init := true;
      end_if;

//--Light and sockets relay control--//
     generalPowerButton(btn := button_24_1);

     if generalPowerButton.shortPress then
        generalPower := true;
     end_if;

     if generalPowerButton.longPress then
        generalPower := false;
     end_if;

     (*MODULE4_OUT.DO5*)
     //electricitySwitch  := generalPower;

     generalPowerObserver(state := generalPower);

//--Global Cache--//
     globalCache( channel := ETH1_uni0 ,
                  codes   := globalCacheCodes);

//--Panel --//
     panel( button[1].btn := MODULE6_IN.DI.DI1,
            button[2].btn := MODULE6_IN.DI.DI2,
            button[3].btn := MODULE6_IN.DI.DI5,
            button[4].btn := MODULE6_IN.DI.DI6,
            button[5].btn := MODULE6_IN.DI.DI4,
            button[6].btn := MODULE6_IN.DI.DI3,
            led[1] => MODULE6_OUT.DOs.DO2,
            led[2] => MODULE6_OUT.DOs.DO3,
            led[3] => MODULE6_OUT.DOs.DO6,
            led[4] => MODULE6_OUT.DOs.DO7,
            led[5] => MODULE6_OUT.DOs.DO5,
            led[6] => MODULE6_OUT.DOs.DO4);

     if generalPowerObserver.rising then
        supervisorAuto01 := true;
        supervisorAuto02 := true;
        supervisorAuto03 := true;
        supervisorAuto04 := true;
        supervisorAuto05 := true;
        supervisorAuto06 := true;
        supervisorAuto07 := true;
        supervisorAuto08 := true;
        //supervisorAuto09 := true;
     end_if;
     if generalPowerObserver.falling then
        supervisorAuto01 := false;
        supervisorAuto02 := false;
        supervisorAuto03 := false;
        supervisorAuto04 := false;
        supervisorAuto05 := false;
        supervisorAuto06 := false;
        supervisorAuto07 := false;
        supervisorAuto08 := false;
        //supervisorAuto09 := false;
     end_if;

END_PROGRAM

(* ---- prgSecurity.ST ---- *)
PROGRAM prgSecurity
  VAR_INPUT
  END_VAR
  VAR_OUTPUT
  END_VAR
  VAR
       security : fbSecuritySystem;
  END_VAR
  VAR_TEMP
  END_VAR

       security(
                 Z1 := true, // door
                 Z2 := true,//(MODULE1_IN.DI0 and MODULE1_IN.DI1 and MODULE1_IN.DI2 and MODULE2_IN.DI.DI1), // entrance/exit zone (hall, kitchen, eatinroom and livingroom)
                 Z3 := (MODULE2_IN.DI.DI4 and MODULE2_IN.DI.DI5 and MODULE1_IN.DI3 and MODULE2_IN.DI.DI2), //bathrooms and bedrooms
                 Z4 := true, //  other sensors, like window contacts and ect.
                 Z5 := true, //  tamper zone

                 arm := security_arm,
                 disarm := security_disarm,
                 alarmReset := security_alarm_reset,

                 securityState => security_state,
                 alarm => security_alarm,
                 ledIndicator => security_led);

      security_arm := false;
      security_alarm_reset:= false;
      security_disarm:= false;

END_PROGRAM

(* ---- prgWardrobeLight.ST ---- *)
PROGRAM prgWardrobeLight
  VAR_INPUT
  END_VAR
  VAR_OUTPUT
  END_VAR
  VAR
      Lamp1     : fbManualRelay;
      button    : fbButtonProcessor;
      Auto      : fbAutoRelay;

      init      : bool;
  END_VAR
  VAR_TEMP
  END_VAR

  if not init then
     r6_1WardrobeLight13_21_auto       := AUTO_MODE_DEFAULT_STATE;
     Auto.timeAfterMotionDetect        := AUTO_MODE_DEFAULT_TIME;
     Auto.Sensor_Motion.mode           := NC;
     Auto.nightMode                    := true;

     init := true;
  end_if;

  button(btn :=MODULE4_IN.DI2 );

  if button.shortPress then
     Lamp1.setState:= not Lamp1.state;
  end_if;

  lamp1( trigButton := r6_1WardrobeLight13_21,
         state      =>  MODULE2_OUT.DOs.DO3
         );

  Auto( Sensor_Motion.state   := MODULE2_IN.DI.DI3,
        autoMode              := r6_1WardrobeLight13_21_auto);

  if Auto.stateChanged OR button.shortPress then
     Lamp1.setState := Auto.state;
  end_if;

END_PROGRAM

(* ---- prgWaterLeakegeControl.ST ---- *)
PROGRAM prgWaterLeakegeControl
  VAR_INPUT
  END_VAR
  VAR_OUTPUT
  END_VAR
  VAR

      waterLeackegeControl: fbWaterLeakegeControl;

      init : bool;

  END_VAR
  VAR_TEMP
  END_VAR

  if not init then
     waterLeackegeControl.config.sensorMode := NO;
     waterLeackegeControl.config.valveMode  := NO;
     waterLeackegeControl.config.timeTreshold := t#4s;
  end_if;

  waterLeackegeControl( sensor    := MODULE7_IN.DI3,
                        openWater := waterOpen,
                        closeWater := waterClose,
                        alarmReset := waterAlarmReset,
                        valve => MODULE4_OUT.DO7,
                        alarm => waterAlarm,
                        waterState := waterState
                        );

  waterOpen  := false;
  waterClose := false;
  waterAlarmReset := false;

  if generalPowerObserver.falling then
     waterState := false;
  end_if;

  if generalPowerObserver.rising then
     waterState := true;
  end_if;

END_PROGRAM
